FUNCTION_BLOCK AnalogInput EXTENDS Component IMPLEMENTS I_AnalogInput, I_AnalogScalable, I_CalibratableLinear
VAR
	Input			 : REFERENCE TO INT;
	Forcible		 : ForcibleInt(_Name);
	_Scale			 : I_AnalogScale;
	_CalibrateLinear : I_CalibrateLinear;
	_CalibrateCustom : I_TransformLRealValue;
END_VAR

VAR
	{attribute 'hide'}
	DefaultScale : AnalogScale;
	{attribute 'hide'}
	DefaultCalibration : Calibrate;
END_VAR

PROPERTY CalibrateCustom : I_TransformLrealValue
SET
_CalibrateCustom := CalibrateCustom;
END_SET
END_PROPERTY

PROPERTY CalibrateLinear : I_CalibrateLinear
GET
CalibrateLinear := _CalibrateLinear;
END_GET
SET
_CalibrateLinear := CalibrateLinear;
END_SET
END_PROPERTY

(*FB_Init is always available implicitly and it is used primarily for initialization.
The return value is not evaluated. For a specific influence, you can also declare the
methods explicitly and provide additional code there with the standard initialization
code. You can evaluate the return value.*)
METHOD FB_Init : BOOL
VAR_INPUT
	(* TRUE: the retain variables are initialized (reset warm / reset cold)*)
	bInitRetains : BOOL;

	(* TRUE: the instance will be copied to the copy code afterward (online change)   *)
	bInCopyCode : BOOL;
	Name		: T_MaxString;
	Input		: REFERENCE TO INT;
END_VAR
_Scale			 := DefaultScale;
_CalibrateLinear := DefaultCalibration;
THIS^.Input		 REF= Input;
END_METHOD

{attribute 'monitoring' := 'call'}
PROPERTY Force : E_ForceState
GET
Force := Forcible.CurrentForceState;
END_GET
SET
VAR
	ForceString : T_MaxString := TO_STRING(Force);
END_VAR
Forcible.SetForceState(Force);
END_SET
END_PROPERTY

PROPERTY ForceValue : INT
GET
ForceValue := Forcible.ForceValue;
END_GET
SET
Forcible.ForceValue := ForceValue;
END_SET
END_PROPERTY

{attribute 'monitoring' := 'call'}
PROPERTY RawValue : INT
GET
Forcible.Input := Input;
RawValue	   := Forcible.Output;
END_GET
END_PROPERTY

PROPERTY Scale : I_AnalogScale
GET
Scale := _Scale;
END_GET
SET
_Scale := Scale;
END_SET
END_PROPERTY

{attribute 'monitoring' := 'call'}
PROPERTY Value : LREAL
GET
IF _CalibrateCustom = 0 THEN
	Value := _CalibrateLinear.Transform(_Scale.Transform(RawValue));
ELSE
	Value := _CalibrateCustom.Transform(_Scale.Transform(RawValue));
END_IF
END_GET
END_PROPERTY

END_FUNCTION_BLOCK

(* stored: Version 1.1.0.1, ProductVersion 3.1.4026.18
   POU AnalogInput: Id {4d270a41-7f74-4fd2-b5a2-ae294d483638}, SpecialFunc None
   Property CalibrateCustom: Id {cf5ffe05-d00e-489d-8c1d-f6fa7d36e68a}
   Set Set: Id {1619d658-d58a-4f65-b1bb-8d984767ac21}
   Property CalibrateLinear: Id {56366c10-60fb-42f7-b82d-be75fc556650}
   Get Get: Id {ed5de5f9-9a64-46c8-bcee-c71dd4ece374}
   Set Set: Id {0d64e2ca-e608-4c2f-bcbd-563d347ae470}
   Method FB_Init: Id {7c54ac1e-4d7c-46ac-8a51-e1a12eeccd69}
   Property Force: Id {afc024e3-a700-419f-96df-f636fdec01d0}
   Get Get: Id {e2f6d948-7d52-4bfb-a9b1-58ed86f5ac94}
   Set Set: Id {8f18cd57-187f-4abb-9a00-0e6cd976a947}
   Property ForceValue: Id {405f6a2d-1d40-4c3c-9fcf-08ec9ab74fba}
   Get Get: Id {6defa823-5945-4ffd-bbf6-7cbc21a8e9d0}
   Set Set: Id {da70e7c7-e92d-41a0-a809-a328f6274423}
   Property RawValue: Id {59ed4d65-3eed-40e7-806c-75b132b200e4}
   Get Get: Id {c298ab88-a4a7-4314-a4c4-072cde6ec9d7}
   Property Scale: Id {c4a5b98b-4797-498d-b7a7-f25e544b4170}
   Get Get: Id {3212b58c-b278-450c-81fc-18864a380a13}
   Set Set: Id {5c9e5b14-d3b5-40ca-a30f-2f78e5110d23}
   Property Value: Id {a78975b4-970f-489d-9eb1-347301f0906a}
   Get Get: Id {1a018181-4754-4469-b9d2-73f0e05aa132} *)
